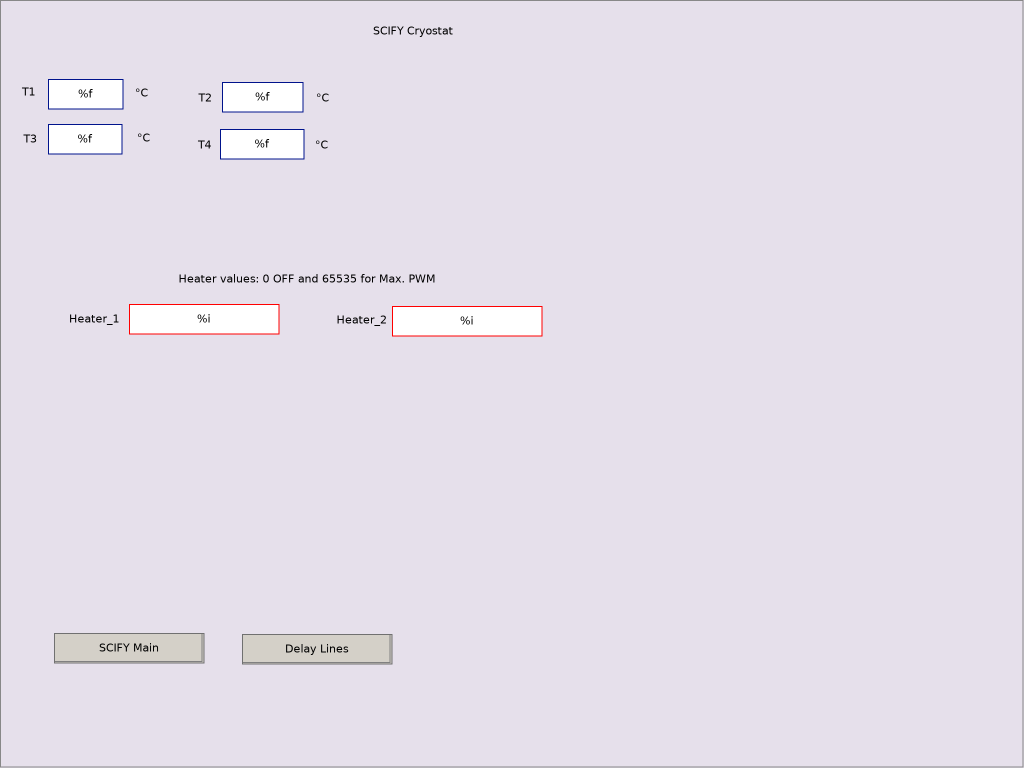
VISUALIZATION SCIFY_Cryo  // 1024x768
    Label (338,6 150x50), "SCIFY Cryostat"
    Textfield (48,79 75x30), "%f", text variable: SCIFY_HMI_Variables.fTemp_1
    Textfield (222,82 81x30), "%f", text variable: SCIFY_HMI_Variables.fTemp_2
    Textfield (48,124 74x30), "%f", text variable: SCIFY_HMI_Variables.fTemp_3
    Textfield (220,129 84x30), "%f", text variable: SCIFY_HMI_Variables.fTemp_4
    Textfield (129,304 150x30), "%i", text variable: SCIFY_HMI_Variables.uiHeater_1
        OnMouseClick: write the text variable via VisuDialogs.Numpad, min 0, max 65535
    Textfield (392,306 150x30), "%i", text variable: SCIFY_HMI_Variables.uiHeater_2
        OnMouseClick: write the text variable via VisuDialogs.Numpad, min 0, max 65535
    Label (19,77 20x30), "T1"
    Label (191,83 29x30), "T2"
    Label (19,124 23x30), "T3"
    Label (196,130 18x30), "T4"
    Label (64,304 61x30), "Heater_1"
    Label (335,305 54x30), "Heater_2"
    Label (122,78 36x30), "°C"
    Label (303,83 36x30), "°C"
    Label (124,123 36x30), "°C"
    Label (302,130 36x30), "°C"
    Label (65,264 484x30), "Heater values: 0 OFF and 65535 for Max. PWM"
    Button (54,633 150x30), "SCIFY Main"
        OnMouseDown: change screen: SCIFY_main
    Button (242,634 150x30), "Delay Lines"
        OnMouseDown: change screen: SCIFY_Delay_Lines
END_VISUALIZATION

(* stored: Version 1.1.0.1, ProductVersion 3.1.4024.12
   Visu SCIFY_Cryo: Id {945a6853-81d5-451b-af1e-ad27577ce62e} *)
